SUBAPPLICATION SubApp_PC_A (* Geraet A (Station 11, 192.168.1.11): SoftKey_F1-Tastendruck und GreenWhiteBackground - 'SUB style', das Protokoll steckt im MyLib::sys-Composite (Softkey_Toggle_RPC_TO_Remote_BG_OPC), nicht in der Resource des Geraets *)
  (* Standard: 61499-2; Description: Copyright (c) 2026 Meisterschulen am Ostbahnhof This program and the accompanying materials are made available under the terms of the Eclipse Public License 2.0 which is available at https://www.eclipse.org/legal/epl-2.0/ SPDX-License-Identifier: EPL-2.0 *)
  (* Version 1.0, 2026-09-02, Franz Höpfinger, Meisterschulen am Ostbahnhof, initial API and implementation and/or initial documentation *)
  PACKAGE subapp::Training_03_OPC_UA_RES;
  IMPORT Uebungen::const::UT::DefaultPool::SoftKey_F1;
  IMPORT VV::const::OPC_UA::myOpcUaAddresses::FF1_TRIGGER_REMOTE_CALL;
  IMPORT VV::const::OPC_UA::myOpcUaAddresses::FF1_STATE_LOCAL_READ;
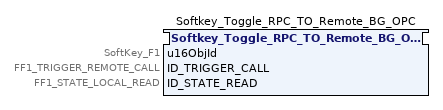
  SUBAPPS
    Softkey_Toggle_RPC_TO_Remote_BG_OPC : MyLib::sys::Softkey_Toggle_RPC_TO_Remote_BG_OPC(u16ObjId := SoftKey_F1, ID_TRIGGER_CALL := FF1_TRIGGER_REMOTE_CALL, ID_STATE_READ := FF1_STATE_LOCAL_READ);
  END_SUBAPPS
END_SUBAPPLICATION
